FUNCTION_BLOCK FB_Dispenser EXTENDS FB_PackML_BaseModule IMPLEMENTS I_Dispenser
VAR
	// Interfaces
	Pump	:	I_Pump;
	Scale	:	I_Scale;
	
	// FBs
	DcPump		: FB_DcPump;
	SerialScale	: FB_SerialScale;
END_VAR

{warning 'Add method implementation '}
METHOD ChangeMode
VAR_INPUT
	Mode	: SPT_BaseTypes.E_PMLUnitMode;
END_VAR
END_METHOD

{warning 'Add method implementation '}
METHOD ChangeState
VAR_INPUT
	State	: SPT_BaseTypes.E_PMLCommand;
END_VAR
END_METHOD

{error 'Add property implementation or delete property to use base implementation'}
PROPERTY CurrentMode : SPT_BaseTypes.E_PMLUnitMode
GET
END_GET
END_PROPERTY

{error 'Add property implementation or delete property to use base implementation'}
PROPERTY CurrentState : SPT_BaseTypes.E_PMLState
GET
END_GET
END_PROPERTY

{warning 'Add method implementation '}
METHOD CyclicLogic
END_METHOD

{warning 'Add property implementation'}
PROPERTY Dispensing : BOOL
GET
END_GET
END_PROPERTY

{warning 'Add property implementation'}
PROPERTY Done : BOOL
GET
END_GET
END_PROPERTY

{warning 'Add method implementation '}
METHOD StartDispense
END_METHOD

METHOD Stop
END_METHOD

{warning 'Add property implementation'}
PROPERTY TargetWeight : LREAL
GET
END_GET
SET
END_SET
END_PROPERTY

END_FUNCTION_BLOCK

(* stored: Version 1.1.0.1
   POU FB_Dispenser: Id {c41dc19d-18c8-416a-bdf6-55f7b512e9fa}, SpecialFunc None
   Method ChangeMode: Id {ae57d5d3-047a-4033-9529-ea645fd3affd}
   Method ChangeState: Id {0779d0e4-e037-4829-a5fc-79ccc358f1df}
   Property CurrentMode: Id {996abd19-e6f0-48fd-8c7b-44e79077ef27}
   Get Get: Id {0c6e7251-28eb-4828-b8d1-0a87c9e0effa}
   Property CurrentState: Id {c4f8866d-7853-44e7-9287-53e037447fdf}
   Get Get: Id {d7d21b1c-5606-4ba7-8782-9c7ac2e0986f}
   Method CyclicLogic: Id {07572f53-0d4a-4171-8afe-15b5f8b0f9d6}
   Property Dispensing: Id {6d2b9f7b-6359-405c-b9ec-8f7410aa8d45}
   Get Get: Id {b4785766-2e72-4600-9375-aefab15567a0}
   Property Done: Id {b0948b1c-3098-4d2b-91cf-ca6aa79a7367}
   Get Get: Id {a4c4d789-6df0-40b0-b637-5aa73cdc84da}
   Method StartDispense: Id {ae324062-b3bd-4131-b4f3-edebd387f563}
   Method Stop: Id {f17e11d8-8278-4919-a3e4-08940dc34e68}
   Property TargetWeight: Id {e01fc650-802b-4b27-9fc8-3cbf080d8d9c}
   Get Get: Id {d29f0bf3-01fc-409a-800c-0cfa643300ee}
   Set Set: Id {e931f160-f032-4882-b42b-9256e975cdaa} *)
